// TIA Portal V20 export
VAR_GLOBAL   // PLC tag table "Default tag table"
   BA030AZSCDR1_Unwinder1_Interface_AddressIn AT %I5114.0 : "PD_TEL105_IN";
   BA030AZSCDR1_Unwinder1_AddressOut AT %Q5114.0 : "PD_TEL105_OUT";
   BA030AZSCDR2_Unwinder2_Actor_Interface_AddressIn AT %I5154.0 : "PD_TEL105_IN";
   BA030AZSCDR2_Unwinder2_Actor_Interface_AddressOut AT %Q5154.0 : "PD_TEL105_OUT";
   BA030AZSCDR5_AnodeMainPnp1AxisX_Actor_Interface_AddressIn AT %I5268.0 : "PD_TEL105_IN";
   BA030AZSCDR5_AnodeMainPnp1AxisX_Actor_Interface_AddressOut AT %Q5268.0 : "PD_TEL105_OUT";
   BA030AZSCDR6_AnodeMainPnp2AxisX_Actor_Interface_AddressIn AT %I5302.0 : "PD_TEL105_IN";
   BA030AZSCDR6_AnodeMainPnp2AxisX_Actor_Interface_AddressOut AT %Q5302.0 : "PD_TEL105_OUT";
   BA030AZSCDR7_CathodeMainPnp1AxisX_Actor_Interface_AddressIn AT %I5336.0 : "PD_TEL105_IN";
   BA030AZSCDR7_CathodeMainPnp1AxisX_Actor_Interface_AddressOut AT %Q5336.0 : "PD_TEL105_OUT";
   BA030AZSCDR8_CathodeMainPnp2AxisX_Actor_Interface_AddressIn AT %I5370.0 : "PD_TEL105_IN";
   BA030AZSCDR8_CathodeMainPnp2AxisX_Actor_Interface_AddressOut AT %Q5370.0 : "PD_TEL105_OUT";
   BA030AZSCDR9_AnodeMainPnp1AxisY_Actor_Interface_AddressIn AT %I5404.0 : "PD_TEL105_IN";
   BA030AZSCDR9_AnodeMainPnp1AxisY_Actor_Interface_AddressOut AT %Q5404.0 : "PD_TEL105_OUT";
   BA030AZSCDR10_AnodeMainPnp1AxisZ_Actor_Interface_AddressIn AT %I5438.0 : "PD_TEL105_IN";
   BA030AZSCDR10_AnodeMainPnp1AxisZ_Actor_Interface_AddressOut AT %Q5438.0 : "PD_TEL105_OUT";
   BA030AZSCDR11_AnodeMainPnp2AxisZ_Actor_Interface_AddressIn AT %I5482.0 : "PD_TEL105_IN";
   BA030AZSCDR11_AnodeMainPnp2AxisZ_Actor_Interface_AddressOut AT %Q5482.0 : "PD_TEL105_OUT";
   BA030AZSCDR12_CathodeMainPnp2AxisZ_Actor_Interface_AddressIn AT %I5516.0 : "PD_TEL105_IN";
   BA030AZSCDR12_CathodeMainPnp2AxisZ_Actor_Interface_AddressOut AT %Q5516.0 : "PD_TEL105_OUT";
   BA030AZSCDR13_CathodeMainPnp1AxisX_Actor_Interface_AddressIn AT %I5560.0 : "PD_TEL105_IN";
   BA030AZSCDR13_CathodeMainPnp1AxisX_Actor_Interface_AddressOut AT %Q5560.0 : "PD_TEL105_OUT";
   BA030AZSCDR14_CathodeMainPnp1AxisZ_Actor_Interface_AddressIn AT %I5604.0 : "PD_TEL105_IN";
   BA030AZSCDR14_CathodeMainPnp1AxisZ_Actor_Interface_AddressOut AT %Q5604.0 : "PD_TEL105_OUT";
   BA030AZSCDR15_AnodeAlignTableAxisU_Actor_Interface_AddressIn AT %I5648.0 : "PD_TEL105_IN";
   BA030AZSCDR15_AnodeAlignTableAxisU_Actor_Interface_AddressOut AT %Q5648.0 : "PD_TEL105_OUT";
   BA030AZSCDR16_AnodeAlignTableAxisV_Actor_Interface_AddressIn AT %I5682.0 : "PD_TEL105_IN";
   BA030AZSCDR16_AnodeAlignTableAxisV_Actor_Interface_AddressOut AT %Q5682.0 : "PD_TEL105_OUT";
   BA030AZSCDR17_AnodeAlignTableAxisW_Actor_Interface_AddressIn AT %I5716.0 : "PD_TEL105_IN";
   BA030AZSCDR17_AnodeAlignTableAxisW_Actor_Interface_AddressOut AT %Q5716.0 : "PD_TEL105_OUT";
   BA030AZSCDR18_CathodeAlignTableAxisU_Actor_Interface_AddressIn AT %I5750.0 : "PD_TEL105_IN";
   BA030AZSCDR18_CathodeAlignTableAxisU_Actor_Interface_AddressOut AT %Q5750.0 : "PD_TEL105_OUT";
   BA030AZSCDR19_CathodeAlignTableAxisV_Actor_Interface_AddressIn AT %I5784.0 : "PD_TEL105_IN";
   BA030AZSCDR19_CathodeAlignTableAxisV_Actor_Interface_AddressOut AT %Q5784.0 : "PD_TEL105_OUT";
   BA030AZSCDR20_CathodeAlignTableAxisW_Actor_Interface_AddressIn AT %I5818.0 : "PD_TEL105_IN";
   BA030AZSCDR20_CathodeAlignTableAxisW_Actor_Interface_AddressOut AT %Q5818.0 : "PD_TEL105_OUT";
   BA030AZSCDR40_JellyRollWinder1AxisY_Actor_Interface_AddressIn AT %I6588.0 : "PD_TEL105_IN";
   BA030AZSCDR40_JellyRollWinder1AxisY_Actor_Interface_AddressOut AT %Q6588.0 : "PD_TEL105_OUT";
   BA030AZSCDR41_JellyRollWinder2AxisY_Actor_Interface_AddressIn AT %I6622.0 : "PD_TEL105_IN";
   BA030AZSCDR41_JellyRollWinder2AxisY_Actor_Interface_AddressOut AT %Q6622.0 : "PD_TEL105_OUT";
   BA030AZSDR1_UnwinderTopAxisB_Actor_Interface_TorqueDataAddressIn AT %I8000.0 : "PD_TEL750_IN";
   BA030AZSDR1_UnwinderTopAxisB_Actor_Interface_TorqueDataAddressOut AT %Q8000.0 : "PD_TEL750_OUT";
   BA030AZSDR4_SepaFeedingRollerAxisB_Actor_Interface_AddressIn AT %I5234.0 : "PD_TEL105_IN";
   BA030AZSDR4_SepaFeedingRollerAxisB_Actor_Interface_AddressOut AT %Q5234.0 : "PD_TEL105_OUT";
   BA030AZSDR4_SepaFeedingRollerAxisB_Actor_Interface_TorqueDataAddressIn AT %I8030.0 : "PD_TEL750_IN";
   BA030AZSDR4_SepaFeedingRollerAxisB_Actor_Interface_TorqueDataAddressOut AT %Q8030.0 : "PD_TEL750_OUT";
   BA030AZSCDR21_FinalRollerFrontAxisX_Actor_Interface_AddressIn AT %I5852.0 : "PD_TEL105_IN";
   BA030AZSCDR21_FinalRollerFrontAxisX_Actor_Interface_AddressOut AT %Q5852.0 : "PD_TEL105_OUT";
   BA030AZSCDR22_FinalRollerRearAxisX_Actor_Interface_AddressIn AT %I5886.0 : "PD_TEL105_IN";
   BA030AZSCDR22_FinalRollerRearAxisX_Actor_Interface_AddressOut AT %Q5886.0 : "PD_TEL105_OUT";
   BA030AZSCDR23_MendrelAnodeFrontAxisY_Actor_Interface_AddressIn AT %I5920.0 : "PD_TEL105_IN";
   BA030AZSCDR23_MendrelAnodeFrontAxisY_Actor_Interface_AddressOut AT %Q5920.0 : "PD_TEL105_OUT";
   BA030AZSCDR24_MendrelAnodeFrontAxisZ_Actor_Interface_AddressIn AT %I5954.0 : "PD_TEL105_IN";
   BA030AZSCDR24_MendrelAnodeFrontAxisZ_Actor_Interface_AddressOut AT %Q5954.0 : "PD_TEL105_OUT";
   BA030AZSCDR25_MendrelAnodeRearAxisY_Actor_Interface_AddressIn AT %I5998.0 : "PD_TEL105_IN";
   BA030AZSCDR25_MendrelAnodeRearAxisY_Actor_Interface_AddressOut AT %Q5998.0 : "PD_TEL105_OUT";
   BA030AZSCDR26_MendrelAnodeRearAxisZ_Actor_Interface_AddressIn AT %I6032.0 : "PD_TEL105_IN";
   BA030AZSCDR26_MendrelAnodeRearAxisZ_Actor_Interface_AddressOut AT %Q6032.0 : "PD_TEL105_OUT";
   BA030AZSCDR27_MendrelCathodeFrontAxisY_Actor_Interface_AddressIn AT %I6076.0 : "PD_TEL105_IN";
   BA030AZSCDR27_MendrelCathodeFrontAxisY_Actor_Interface_AddressOut AT %Q6076.0 : "PD_TEL105_OUT";
   BA030AZSCDR28_MendrelCathodeFrontAxisZ_Actor_Interface_AddressIn AT %I6110.0 : "PD_TEL105_IN";
   BA030AZSCDR28_MendrelCathodeFrontAxisZ_Actor_Interface_AddressOut AT %Q6110.0 : "PD_TEL105_OUT";
   BA030AZSCDR29_MendrelCathodeRearAxisY_Actor_Interface_AddressIn AT %I6154.0 : "PD_TEL105_IN";
   BA030AZSCDR29_MendrelCathodeRearAxisY_Actor_Interface_AddressOut AT %Q6154.0 : "PD_TEL105_OUT";
   BA030AZSCDR30_MendrelCathodeRearAxisZ_Actor_Interface_AddressIn AT %I6188.0 : "PD_TEL105_IN";
   BA030AZSCDR30_MendrelCathodeRearAxisZ_Actor_Interface_AddressOut AT %Q6188.0 : "PD_TEL105_OUT";
   BA030AZSCDR31_StackTableAxisZ_Actor_Interface_AddressIn AT %I6232.0 : "PD_TEL105_IN";
   BA030AZSCDR31_StackTableAxisZ_Actor_Interface_AddressOut AT %Q6232.0 : "PD_TEL105_OUT";
   BA030AZSCDR32_StackTableOutFrontAxisZ_Actor_Interface_AddressIn AT %I6276.0 : "PD_TEL105_IN";
   BA030AZSCDR32_StackTableOutFrontAxisZ_Actor_Interface_AddressOut AT %Q6276.0 : "PD_TEL105_OUT";
   BA030AZSCDR33_StackTableOutRearAxisZ_Actor_Interface_AddressIn AT %I6320.0 : "PD_TEL105_IN";
   BA030AZSCDR33_StackTableOutRearAxisZ_Actor_Interface_AddressOut AT %Q6320.0 : "PD_TEL105_OUT";
   BA030AZSCDR34_SepaClampnCutterAxisX_Actor_Interface_AddressIn AT %I6364.0 : "PD_TEL105_IN";
   BA030AZSCDR34_SepaClampnCutterAxisX_Actor_Interface_AddressOut AT %Q6364.0 : "PD_TEL105_OUT";
   BA030AZSCDR35_SepaClampnCutterAxisZ_Actor_Interface_AddressIn AT %I6398.0 : "PD_TEL105_IN";
   BA030AZSCDR35_SepaClampnCutterAxisZ_Actor_Interface_AddressOut AT %Q6398.0 : "PD_TEL105_OUT";
   BA030AZSCDR36_SepaGripperAxisX_Actor_Interface_AddressIn AT %I6442.0 : "PD_TEL105_IN";
   BA030AZSCDR36_SepaGripperAxisX_Actor_Interface_AddressOut AT %Q6442.0 : "PD_TEL105_OUT";
   BA030AZSCDR37_SepaGripperAxisZ_Actor_Interface_AddressIn AT %I6476.0 : "PD_TEL105_IN";
   BA030AZSCDR37_SepaGripperAxisZ_Actor_Interface_AddressOut AT %Q6476.0 : "PD_TEL105_OUT";
   BA030AZSCDR38_SepaGripperAxisC_Actor_Interface_AddressIn AT %I6520.0 : "PD_TEL105_IN";
   BA030AZSCDR38_SepaGripperAxisC_Actor_Interface_AddressOut AT %Q6520.0 : "PD_TEL105_OUT";
   BA030AZSCDR39_JRWinderRearAxisY_Actor_Interface_AddressIn AT %I6554.0 : "PD_TEL105_IN";
   BA030AZSCDR39_JRWinderRearAxisY_Actor_Interface_AddressOut AT %Q6554.0 : "PD_TEL105_OUT";
   BA030AZSDR3_CompensatorAxisX_Actor_Interface_AddressIn AT %I5194.0 : "PD_TEL105_IN";
   BA030AZSDR3_CompensatorAxisX_Actor_Interface_AddressOut AT %Q5194.0 : "PD_TEL105_OUT";
   BA030AZSCDR39_JRWinderRearAxisY_Actor_Interface_TorqueDataAddressIn AT %I8380.0 : "PD_TEL750_IN";
   BA030AZSCDR39_JRWinderRearAxisY_Actor_Interface_TorqueDataAddressOut AT %Q8380.0 : "PD_TEL750_OUT";
   BA030AZSCDR6_AnodeMainPnp2AxisX_Actor_Interface_TorqueDataAddressIn AT %I8050.0 : "PD_TEL750_IN";
   BA030AZSCDR6_AnodeMainPnp2AxisX_Actor_Interface_TorqueDataAddressOut AT %Q8050.0 : "PD_TEL750_OUT";
   BA030AZSCDR11_AnodeMainPnp1AxisY_Actor_Interface_TorqueDataAddressIn AT %I8100.0 : "PD_TEL750_IN";
   BA030AZSCDR11_AnodeMainPnp1AxisY_Actor_Interface_TorqueDataAddressOut AT %Q8100.0 : "PD_TEL750_OUT";
   BA030AZSCDR12_AnodeMainPnp1AxisZ_Actor_Interface_TorqueDataAddressIn AT %I8110.0 : "PD_TEL750_IN";
   BA030AZSCDR12_AnodeMainPnp1AxisZ_Actor_Interface_TorqueDataAddressOut AT %Q8110.0 : "PD_TEL750_OUT";
   BA030AZSCDR14_AnodeMainPnp2AxisZ_Actor_Interface_TorqueDataAddressIn AT %I8130.0 : "PD_TEL750_IN";
   BA030AZSCDR14_AnodeMainPnp2AxisZ_Actor_Interface_TorqueDataAddressOut AT %Q8130.0 : "PD_TEL750_OUT";
   BA030AZSCDR15_AnodeAlignTableAxisX_Actor_Interface_TorqueDataAddressIn AT %I8140.0 : "PD_TEL750_IN";
   BA030AZSCDR15_AnodeAlignTableAxisX_Actor_Interface_TorqueDataAddressOut AT %Q8140.0 : "PD_TEL750_OUT";
   BA030AZSCDR16_AnodeAlignTableAxisY1_Actor_Interface_TorqueDataAddressIn AT %I8150.0 : "PD_TEL750_IN";
   BA030AZSCDR16_AnodeAlignTableAxisY1_Actor_Interface_TorqueDataAddressOut AT %Q8150.0 : "PD_TEL750_OUT";
   BA030AZSCDR17_AnodeAlignTableAxisY2_Actor_Interface_TorqueDataAddressIn AT %I8160.0 : "PD_TEL750_IN";
   BA030AZSCDR17_AnodeAlignTableAxisY2_Actor_Interface_TorqueDataAddressOut AT %Q8160.0 : "PD_TEL750_OUT";
   BA030AZSCDR7_CathodeMainPnp1AxisX_Actor_Interface_TorqueDataAddressIn AT %I8060.0 : "PD_TEL750_IN";
   BA030AZSCDR7_CathodeMainPnp1AxisX_Actor_Interface_TorqueDataAddressOut AT %Q8060.0 : "PD_TEL750_OUT";
   BA030AZSCDR8_CathodeMainPnp2AxisX_Actor_Interface_TorqueDataAddressIn AT %I8070.0 : "PD_TEL750_IN";
   BA030AZSCDR8_CathodeMainPnp2AxisX_Actor_Interface_TorqueDataAddressOut AT %Q8070.0 : "PD_TEL750_OUT";
   BA030AZSCDR9_CathodeMainPnp1AxisY_Actor_Interface_TorqueDataAddressIn AT %I8080.0 : "PD_TEL750_IN";
   BA030AZSCDR9_CathodeMainPnp1AxisY_Actor_Interface_TorqueDataAddressOut AT %Q8080.0 : "PD_TEL750_OUT";
   BA030AZSCDR13_CathodeMainPnp2AxisZ_Actor_Interface_TorqueDataAddressIn AT %I8120.0 : "PD_TEL750_IN";
   BA030AZSCDR13_CathodeMainPnp2AxisZ_Actor_Interface_TorqueDataAddressOut AT %Q8120.0 : "PD_TEL750_OUT";
   BA030AZSCDR18_CathodeAlignTableAxisX_Actor_Interface_TorqueDataAddressIn AT %I8170.0 : "PD_TEL750_IN";
   BA030AZSCDR18_CathodeAlignTableAxisX_Actor_Interface_TorqueDataAddressOut AT %Q8170.0 : "PD_TEL750_OUT";
   BA030AZSCDR19_CathodeAlignTableAxisY1_Actor_Interface_TorqueDataAddressIn AT %I8180.0 : "PD_TEL750_IN";
   BA030AZSCDR19_CathodeAlignTableAxisY1_Actor_Interface_TorqueDataAddressOut AT %Q8180.0 : "PD_TEL750_OUT";
   BA030AZSCDR20_CathodeAlignTableAxisY2_Actor_Interface_TorqueDataAddressIn AT %I8190.0 : "PD_TEL750_IN";
   BA030AZSCDR20_CathodeAlignTableAxisY2_Actor_Interface_TorqueDataAddressOut AT %Q8190.0 : "PD_TEL750_OUT";
   BA030AZSCDR21_FinalRollerFrontAxisX_Actor_Interface_TorqueDataAddressIn AT %I8200.0 : "PD_TEL750_IN";
   BA030AZSCDR21_FinalRollerFrontAxisX_Actor_Interface_TorqueDataAddressOut AT %Q8200.0 : "PD_TEL750_OUT";
   BA030AZSCDR22_FinalRollerRearAxisX_Actor_Interface_TorqueDataAddressIn AT %I8210.0 : "PD_TEL750_IN";
   BA030AZSCDR22_FinalRollerRearAxisX_Actor_Interface_TorqueDataAddressOut AT %Q8210.0 : "PD_TEL750_OUT";
   BA030AZSCDR23_MendrelAnodeFrontAxisY_Actor_Interface_TorqueDataAddressIn AT %I8220.0 : "PD_TEL750_IN";
   BA030AZSCDR23_MendrelAnodeFrontAxisY_Actor_Interface_TorqueDataAddressOut AT %Q8220.0 : "PD_TEL750_OUT";
   BA030AZSCDR24_MendrelAnodeFrontAxisZ_Actor_Interface_TorqueDataAddressIn AT %I8230.0 : "PD_TEL750_IN";
   BA030AZSCDR24_MendrelAnodeFrontAxisZ_Actor_Interface_TorqueDataAddressOut AT %Q8230.0 : "PD_TEL750_OUT";
   BA030AZSCDR25_MendrelAnodeRearAxisY_Actor_Interface_TorqueDataAddressIn AT %I8240.0 : "PD_TEL750_IN";
   BA030AZSCDR25_MendrelAnodeRearAxisY_Actor_Interface_TorqueDataAddressOut AT %Q8240.0 : "PD_TEL750_OUT";
   BA030AZSCDR26_MendrelAnodeRearAxisZ_Actor_Interface_TorqueDataAddressIn AT %I8250.0 : "PD_TEL750_IN";
   BA030AZSCDR26_MendrelAnodeRearAxisZ_Actor_Interface_TorqueDataAddressOut AT %Q8250.0 : "PD_TEL750_OUT";
   BA030AZSCDR27_MendrelCathodeFrontAxisY_Actor_Interface_TorqueDataAddressIn AT %I8260.0 : "PD_TEL750_IN";
   BA030AZSCDR27_MendrelCathodeFrontAxisY_Actor_Interface_TorqueDataAddressOut AT %Q8260.0 : "PD_TEL750_OUT";
   BA030AZSCDR28_MendrelCathodeFrontAxisZ_Actor_Interface_TorqueDataAddressIn AT %I8270.0 : "PD_TEL750_IN";
   BA030AZSCDR28_MendrelCathodeFrontAxisZ_Actor_Interface_TorqueDataAddressOut AT %Q8270.0 : "PD_TEL750_OUT";
   BA030AZSCDR29_MendrelCathodeRearAxisY_Actor_Interface_TorqueDataAddressIn AT %I8280.0 : "PD_TEL750_IN";
   BA030AZSCDR29_MendrelCathodeRearAxisY_Actor_Interface_TorqueDataAddressOut AT %Q8280.0 : "PD_TEL750_OUT";
   BA030AZSCDR30_MendrelCathodeRearAxisZ_Actor_Interface_TorqueDataAddressIn AT %I8290.0 : "PD_TEL750_IN";
   BA030AZSCDR30_MendrelCathodeRearAxisZ_Actor_Interface_TorqueDataAddressOut AT %Q8290.0 : "PD_TEL750_OUT";
   BA030AZSCDR31_StackTableAxisZ_Actor_Interface_TorqueDataAddressIn AT %I8300.0 : "PD_TEL750_IN";
   BA030AZSCDR31_StackTableAxisZ_Actor_Interface_TorqueDataAddressOut AT %Q8300.0 : "PD_TEL750_OUT";
   BA030AZSCDR32_StackTableOutFrontAxisZ_Actor_Interface_TorqueDataAddressIn AT %I8310.0 : "PD_TEL750_IN";
   BA030AZSCDR32_StackTableOutFrontAxisZ_Actor_Interface_TorqueDataAddressOut AT %Q8310.0 : "PD_TEL750_OUT";
   BA030AZSCDR33_StackTableOutRearAxisZ_Actor_Interface_TorqueDataAddressIn AT %I8320.0 : "PD_TEL750_IN";
   BA030AZSCDR33_StackTableOutRearAxisZ_Actor_Interface_TorqueDataAddressOut AT %Q8320.0 : "PD_TEL750_OUT";
   BA030AZSCDR34_SepaClampnCutterAxisX_Actor_Interface_TorqueDataAddressIn AT %I8330.0 : "PD_TEL750_IN";
   BA030AZSCDR34_SepaClampnCutterAxisX_Actor_Interface_TorqueDataAddressOut AT %Q8330.0 : "PD_TEL750_OUT";
   BA030AZSCDR35_SepaClampnCutterAxisZ_Actor_Interface_TorqueDataAddressIn AT %I8340.0 : "PD_TEL750_IN";
   BA030AZSCDR35_SepaClampnCutterAxisZ_Actor_Interface_TorqueDataAddressOut AT %Q8340.0 : "PD_TEL750_OUT";
   BA030AZSCDR36_SepaGripperAxisX_Actor_Interface_TorqueDataAddressIn AT %I8350.0 : "PD_TEL750_IN";
   BA030AZSCDR36_SepaGripperAxisX_Actor_Interface_TorqueDataAddressOut AT %Q8350.0 : "PD_TEL750_OUT";
   BA030AZSCDR37_SepaGripperAxisZ_Actor_Interface_TorqueDataAddressIn AT %I8360.0 : "PD_TEL750_IN";
   BA030AZSCDR37_SepaGripperAxisZ_Actor_Interface_TorqueDataAddressOut AT %Q8360.0 : "PD_TEL750_OUT";
   BA030AZSCDR38_SepaGripperAxisC_Actor_Interface_TorqueDataAddressIn AT %I8370.0 : "PD_TEL750_IN";
   BA030AZSCDR38_SepaGripperAxisC_Actor_Interface_TorqueDataAddressOut AT %Q8370.0 : "PD_TEL750_OUT";
   BA030AZSCDR40_JRWinderFrontAxisY_Actor_Interface_TorqueDataAddressIn AT %I8390.0 : "PD_TEL750_IN";
   BA030AZSCDR40_JRWinderFrontAxisY_Actor_Interface_TorqueDataAddressOut AT %Q8390.0 : "PD_TEL750_OUT";
   BA030AZSCDR41_JRWinderAxisB_Actor_Interface_TorqueDataAddressIn AT %I8400.0 : "PD_TEL750_IN";
   BA030AZSCDR41_JRWinderAxisB_Actor_Interface_TorqueDataAddressOut AT %Q8400.0 : "PD_TEL750_OUT";
   BA030AZSCDR10_CathodeMainPnp1AxisZ_Actor_Interface_TorqueDataAddressIn AT %I8090.0 : "PD_TEL750_IN";
   BA030AZSCDR10_CathodeMainPnp1AxisZ_Actor_Interface_TorqueDataAddressOut AT %Q8090.0 : "PD_TEL750_OUT";
   BA030AZSDR2_UnwinderBottomAxisB_Actor_Interface_TorqueDataAddressIn AT %I8010.0 : "PD_TEL750_IN";
   BA030AZSDR2_UnwinderBottomAxisB_Actor_Interface_TorqueDataAddressOut AT %Q8010.0 : "PD_TEL750_OUT";
   BA030AZSDR3_CompensatorAxisX_Actor_Interface_TorqueDataAddressIn AT %I8020.0 : "PD_TEL750_IN";
   BA030AZSDR3_CompensatorAxisX_Actor_Interface_TorqueDataAddressOut AT %Q8020.0 : "PD_TEL750_OUT";
   BA030AZSCDR5_AnodeMainPnp1AxisX_Actor_Interface_TorqueDataAddressIn AT %I8040.0 : "PD_TEL750_IN";
   BA030AZSCDR5_AnodeMainPnp1AxisX_Actor_Interface_TorqueDataAddressOut AT %Q8040.0 : "PD_TEL750_OUT";
END_VAR
